// TwinCAT 3 PLC project CNM_RecipeHandling
// Title: CNM_RecipeHandling
// Company: ekvip automation GmbH
// Author: tsch
// ProjectVersion: 0.1.1.0
// Description: This is a TwinCAT 3 library for recipe handling and machine settings. It is intended to be used with CNM HMI framework to store and load parameters.
// ProgramVersion: 3.1.4026.19
// libraries:
//   Tc2_Utilities, * (Beckhoff Automation GmbH)
// project tree:
//   Functions/ CalculateVelocity.TcPOU, ConvertAngle.TcPOU, ConvertAngularVelocity.TcPOU, ConvertArea.TcPOU, ConvertDuration.TcPOU, ConvertLength.TcPOU, ConvertVelocity.TcPOU, ConvertPressure.TcPOU, ConvertTemperature.TcPOU, ConvertVolume.TcPOU, ConvertWeight.TcPOU, FastPow10.TcPOU
//   Functions/Helper/ CheckValueIsANumber.TcPOU
//   Project Information/ F_GetCompany.TcPOU, F_GetTitle.TcPOU, F_GetVersion.TcPOU
//   Types/ Angle.TcDUT, AngularVelocity.TcDUT, Area.TcDUT, BaseParameter.TcDUT, Duration.TcDUT, Length.TcDUT, MetricParameter.TcDUT, Pressure.TcDUT, SiDefaultParameter.TcDUT, Temperature.TcDUT, Velocity.TcDUT, Volume.TcDUT, Weight.TcDUT
//   Types/Units/ AngleUnit.TcDUT, AreaUnit.TcDUT, LengthUnit.TcDUT, DurationUnit.TcDUT, MetricPrefixes.TcDUT, PressureUnit.TcDUT, TemperatureUnit.TcDUT, UnitString.TcDUT, VolumeUnit.TcDUT, WeightUnit.TcDUT
//   Version/ Global_Version.TcGVL

// ---- Types/Angle.TcDUT
(*

## Short summary

A datatype for angles based on angular units. It can be converted to other units with the function CNM_RecipeHandling.ConvertAngle.

.. <legal notes>

legal notes
=================
| SPDX-FileCopyrightText: © 2025 ekvip automation GmbH <info@ekvip.de>
| SPDX-License-Identifier: Apache-2.0
| For details check: Apache-2.0_

.. _Apache-2.0: https://www.apache.org/licenses/LICENSE-2.0

.. </legal notes>	

*)

TYPE Angle EXTENDS BaseParameter:
STRUCT
	(* the angular unit *)
	unit :AngleUnit := AngleUnit.RADIANS;
END_STRUCT
END_TYPE

// ---- Types/AngularVelocity.TcDUT
(*

## Short summary

A datatype for angular velocities based on physical units.

.. <legal notes>

legal notes
=================
| SPDX-FileCopyrightText: © 2025 ekvip automation GmbH <info@ekvip.de>
| SPDX-License-Identifier: Apache-2.0
| For details check: Apache-2.0_

.. _Apache-2.0: https://www.apache.org/licenses/LICENSE-2.0

.. </legal notes>	

*)

TYPE AngularVelocity EXTENDS BaseParameter:
STRUCT
	angularDistanceUnit :AngleUnit := AngleUnit.TURNS;
	timeUnit :DurationUnit := DurationUnit.MINUTE;
	timePrefix :MetricPrefixes := MetricPrefixes.NONE;
END_STRUCT
END_TYPE

// ---- Types/Area.TcDUT
(*

## Short summary

A datatype for areas based on physical units. It can be converted to other units with the function CNM_RecipeHandling.ConvertArea. 

.. <legal notes>

legal notes
=================
| SPDX-FileCopyrightText: © 2025 ekvip automation GmbH <info@ekvip.de>
| SPDX-License-Identifier: Apache-2.0
| For details check: Apache-2.0_

.. _Apache-2.0: https://www.apache.org/licenses/LICENSE-2.0

.. </legal notes>	

*)

TYPE Area EXTENDS MetricParameter:
STRUCT
	(* the area unit *)
	unit :AreaUnit := AreaUnit.SQUARE_METER;
END_STRUCT
END_TYPE

// ---- Types/BaseParameter.TcDUT
(*

## Short summary

A basic datatype for physical parameters. It has just a value. 

.. <legal notes>

legal notes
=================
| SPDX-FileCopyrightText: © 2025 ekvip automation GmbH <info@ekvip.de>
| SPDX-License-Identifier: Apache-2.0
| For details check: Apache-2.0_

.. _Apache-2.0: https://www.apache.org/licenses/LICENSE-2.0

.. </legal notes>	

*)

TYPE BaseParameter :
STRUCT
	value :LREAL := 0.0;
END_STRUCT
END_TYPE

// ---- Types/Duration.TcDUT
(*

## Short summary

A datatype for durations based on physical time units. It can be converted to other units with the function CNM_RecipeHandling.ConvertDuration. 

.. <legal notes>

legal notes
=================
| SPDX-FileCopyrightText: © 2025 ekvip automation GmbH <info@ekvip.de>
| SPDX-License-Identifier: Apache-2.0
| For details check: Apache-2.0_

.. _Apache-2.0: https://www.apache.org/licenses/LICENSE-2.0

.. </legal notes>	

*)

TYPE Duration EXTENDS MetricParameter :
STRUCT
	(* the time unit *)
	unit :DurationUnit := DurationUnit.SECONDS;
END_STRUCT
END_TYPE

// ---- Types/Length.TcDUT
(*

## Short summary

A datatype for distances based on physical length units. It can be converted to other units with the function CNM_RecipeHandling.ConvertLength. 

.. <legal notes>

legal notes
=================
| SPDX-FileCopyrightText: © 2025 ekvip automation GmbH <info@ekvip.de>
| SPDX-License-Identifier: Apache-2.0
| For details check: Apache-2.0_

.. _Apache-2.0: https://www.apache.org/licenses/LICENSE-2.0

.. </legal notes>	

*)

TYPE Length EXTENDS MetricParameter:
STRUCT
	(* the length unit *)
	unit :LengthUnit := LengthUnit.METER;
END_STRUCT
END_TYPE

// ---- Types/MetricParameter.TcDUT
(*

## Short summary

A basic datatype for metrical physical parameters. It extends the CNM_RecipeHandling.BaseParameter with a metric prefix. 

.. <legal notes>

legal notes
=================
| SPDX-FileCopyrightText: © 2025 ekvip automation GmbH <info@ekvip.de>
| SPDX-License-Identifier: Apache-2.0
| For details check: Apache-2.0_

.. _Apache-2.0: https://www.apache.org/licenses/LICENSE-2.0

.. </legal notes>	

*)

TYPE MetricParameter EXTENDS BaseParameter :
STRUCT
	prefix :MetricPrefixes := MetricPrefixes.NONE;
END_STRUCT
END_TYPE

// ---- Types/Pressure.TcDUT
(*

## Short summary

A datatype for pressures based on physical units. It can be converted to other units with the function CNM_RecipeHandling.ConvertPressure. 

.. <legal notes>

legal notes
=================
| SPDX-FileCopyrightText: © 2025 ekvip automation GmbH <info@ekvip.de>
| SPDX-License-Identifier: Apache-2.0
| For details check: Apache-2.0_

.. _Apache-2.0: https://www.apache.org/licenses/LICENSE-2.0

.. </legal notes>	

*)

TYPE Pressure EXTENDS MetricParameter :
STRUCT
	unit :PressureUnit := PressureUnit.PASCAL;
END_STRUCT
END_TYPE

// ---- Types/SiDefaultParameter.TcDUT
(*

## Short summary

A datatype for temperatures based on temperature scales. It can be converted to other units with the function CNM_RecipeHandling.ConvertTemperature. 

.. <legal notes>

legal notes
=================
| SPDX-FileCopyrightText: © 2025 ekvip automation GmbH <info@ekvip.de>
| SPDX-License-Identifier: Apache-2.0
| For details check: Apache-2.0_

.. _Apache-2.0: https://www.apache.org/licenses/LICENSE-2.0

.. </legal notes>	

*)

TYPE SiDefaultParameter EXTENDS MetricParameter :
STRUCT
	unit :UnitString;
END_STRUCT
END_TYPE

// ---- Types/Temperature.TcDUT
(*

## Short summary

A datatype for temperatures based on temperature scales. It can be converted to other units with the function CNM_RecipeHandling.ConvertTemperature. 

.. <legal notes>

legal notes
=================
| SPDX-FileCopyrightText: © 2025 ekvip automation GmbH <info@ekvip.de>
| SPDX-License-Identifier: Apache-2.0
| For details check: Apache-2.0_

.. _Apache-2.0: https://www.apache.org/licenses/LICENSE-2.0

.. </legal notes>	

*)

TYPE Temperature EXTENDS BaseParameter:
STRUCT
	(* the temperature scale *)
	unit :TemperatureUnit := TemperatureUnit.KELVIN;
END_STRUCT
END_TYPE

// ---- Types/Units/AngleUnit.TcDUT
(*

## Short summary

This enumeration contains common angular units including radians, degrees, arc minutes, and arc seconds.

.. <legal notes>

legal notes
=================
| SPDX-FileCopyrightText: © 2025 ekvip automation GmbH <info@ekvip.de>
| SPDX-License-Identifier: Apache-2.0
| For details check: Apache-2.0_

.. _Apache-2.0: https://www.apache.org/licenses/LICENSE-2.0

.. </legal notes>	

*)

{attribute 'qualified_only'}
{attribute 'to_string'}
TYPE AngleUnit :
(
	RADIANS := 0,
	DEGREES,
	ARC_MINUTES,
	ARC_SECONDS,
	GRADIANS,
	TURNS
);
END_TYPE

// ---- Types/Units/AreaUnit.TcDUT
(*

## Short summary

This enumeration contains common physical area units.

.. <legal notes>

legal notes
=================
| SPDX-FileCopyrightText: © 2025 ekvip automation GmbH <info@ekvip.de>
| SPDX-License-Identifier: Apache-2.0
| For details check: Apache-2.0_

.. _Apache-2.0: https://www.apache.org/licenses/LICENSE-2.0

.. </legal notes>	

*)
{attribute 'qualified_only'}
{attribute 'to_string'}
TYPE AreaUnit :
(
	SQUARE_METER := 0,
	US_SQUARE_INCH,
	US_SQUARE_FOOT,
	US_SQUARE_YARD,
	US_ACRE,
	HECTARE
);
END_TYPE

// ---- Types/Units/LengthUnit.TcDUT
(*

## Short summary

This enumeration contains common physical length units.

.. <legal notes>

legal notes
=================
| SPDX-FileCopyrightText: © 2025 ekvip automation GmbH <info@ekvip.de>
| SPDX-License-Identifier: Apache-2.0
| For details check: Apache-2.0_

.. _Apache-2.0: https://www.apache.org/licenses/LICENSE-2.0

.. </legal notes>	

*)

{attribute 'qualified_only'}
{attribute 'to_string'}
TYPE LengthUnit :
(
	METER := 0,
	US_MIL,
	US_INCH,
	US_FOOT,
	US_YARD,
	US_MILE	
);
END_TYPE

// ---- Types/Units/DurationUnit.TcDUT
(*

## Short summary

This enumeration contains common physical time units.

.. <legal notes>

legal notes
=================
| SPDX-FileCopyrightText: © 2025 ekvip automation GmbH <info@ekvip.de>
| SPDX-License-Identifier: Apache-2.0
| For details check: Apache-2.0_

.. _Apache-2.0: https://www.apache.org/licenses/LICENSE-2.0

.. </legal notes>	

*)

{attribute 'qualified_only'}
{attribute 'to_string'}
TYPE DurationUnit :
(
	SECONDS := 0,
	MINUTE,
	HOUR,
	DAY,
	WEEK	
);
END_TYPE

// ---- Types/Units/MetricPrefixes.TcDUT
(*

## Short summary

This is an enumeration for metric prefixes. The value after an enum entry corresponds to the power of ten of the respective prefix. 

.. <legal notes>

legal notes
=================
| SPDX-FileCopyrightText: © 2025 ekvip automation GmbH <info@ekvip.de>
| SPDX-License-Identifier: Apache-2.0
| For details check: Apache-2.0_

.. _Apache-2.0: https://www.apache.org/licenses/LICENSE-2.0

.. </legal notes>	

*)

{attribute 'qualified_only'}
{attribute 'to_string'}
TYPE MetricPrefixes :
(
	QUECTO := -30,
	RONTO := -27 ,
	YOCTO := -24 ,
	ZEPTO := -21 ,
	ATTO := -18  ,
	FEMTO := -15 ,
	PICO := -12  ,
	NANO := -9   ,
	MICRO := -6  ,
	MILLI := -3  ,
	CENTI := -2  ,
	DECI := -1   ,
	NONE := 0    ,
	DEKA := 1    ,
	HECTO := 2   ,
	KILO := 3    ,
	MEGA := 6    ,
	GIGA := 9    ,
	TERA := 12   ,
	PETA := 15   ,
	EXA := 18    ,
	ZETTA := 21  ,
	YOTTA := 24  ,
	RONNA := 27  ,
	QUETTA := 30 
) INT ;
END_TYPE

// ---- Types/Units/PressureUnit.TcDUT
(*

## Short summary

This enumeration contains common physical pressure units.

.. <legal notes>

legal notes
=================
| SPDX-FileCopyrightText: © 2025 ekvip automation GmbH <info@ekvip.de>
| SPDX-License-Identifier: Apache-2.0
| For details check: Apache-2.0_

.. _Apache-2.0: https://www.apache.org/licenses/LICENSE-2.0

.. </legal notes>	

*)

{attribute 'qualified_only'}
{attribute 'to_string'}
TYPE PressureUnit :
(
	PASCAL := 0,
	BAR,
	(* pound per square inch *)
	PSI
);
END_TYPE

// ---- Types/Units/TemperatureUnit.TcDUT
(*

## Short summary

This enumeration contains common temperature scales.

.. <legal notes>

legal notes
=================
| SPDX-FileCopyrightText: © 2025 ekvip automation GmbH <info@ekvip.de>
| SPDX-License-Identifier: Apache-2.0
| For details check: Apache-2.0_

.. _Apache-2.0: https://www.apache.org/licenses/LICENSE-2.0

.. </legal notes>	

*)

{attribute 'qualified_only'}
{attribute 'to_string'}
TYPE TemperatureUnit :
(
	KELVIN := 0,
	DEGREE_CELSIUS,
	DEGREE_FAHRENHEIT
);
END_TYPE

// ---- Types/Units/UnitString.TcDUT
(*

## Short summary

The UnitString is an alias for a string with a limited amount of characters. 

.. <legal notes>

legal notes
=================
| SPDX-FileCopyrightText: © 2025 ekvip automation GmbH <info@ekvip.de>
| SPDX-License-Identifier: Apache-2.0
| For details check: Apache-2.0_

.. _Apache-2.0: https://www.apache.org/licenses/LICENSE-2.0

.. </legal notes>	

*)

TYPE UnitString : STRING(10); END_TYPE

// ---- Types/Units/VolumeUnit.TcDUT
(*

## Short summary

This enumeration contains common physical volume units.

.. <legal notes>

legal notes
=================
| SPDX-FileCopyrightText: © 2025 ekvip automation GmbH <info@ekvip.de>
| SPDX-License-Identifier: Apache-2.0
| For details check: Apache-2.0_

.. _Apache-2.0: https://www.apache.org/licenses/LICENSE-2.0

.. </legal notes>	

*)

{attribute 'qualified_only'}
{attribute 'strict'}
{attribute 'to_string'}
TYPE VolumeUnit :
(
	CUBIC_METER := 0,
	LITER,
	US_CUBIC_INCH,
	US_CUBIC_FOOT,
	US_CUBIC_YARD,
	US_FLUID_OUNCE,
	US_PINT,
	US_GALLON,
	US_BARREL,
	US_OIL_BARREL,
	US_DRY_PINT,
	US_DRY_GALLON,
	US_DRY_BARREL
);
END_TYPE

// ---- Types/Units/WeightUnit.TcDUT
(*

## Short summary

This enumeration contains common physical weight units. The US units are based on the Avoirdupois measurement system.

.. <legal notes>

legal notes
=================
| SPDX-FileCopyrightText: © 2025 ekvip automation GmbH <info@ekvip.de>
| SPDX-License-Identifier: Apache-2.0
| For details check: Apache-2.0_

.. _Apache-2.0: https://www.apache.org/licenses/LICENSE-2.0

.. </legal notes>	

*)


{attribute 'qualified_only'}
{attribute 'to_string'}
TYPE WeightUnit :
(
	GRAM := 0,
	TON,
	US_GRAIN,
	US_DRAM,
	US_OUNCE,
	US_POUND,
	US_TON
);
END_TYPE

// ---- Types/Velocity.TcDUT
(*

## Short summary

A datatype for velocities based on physical units. It can be converted to other units with the function CNM_RecipeHandling.ConvertVelocity.

.. <legal notes>

legal notes
=================
| SPDX-FileCopyrightText: © 2025 ekvip automation GmbH <info@ekvip.de>
| SPDX-License-Identifier: Apache-2.0
| For details check: Apache-2.0_

.. _Apache-2.0: https://www.apache.org/licenses/LICENSE-2.0

.. </legal notes>	

*)

TYPE Velocity EXTENDS BaseParameter:
STRUCT
	distanceUnit :LengthUnit := LengthUnit.METER;
	distancePrefix :MetricPrefixes := MetricPrefixes.NONE;
	timeUnit :DurationUnit := DurationUnit.SECONDS;
	timePrefix :MetricPrefixes := MetricPrefixes.NONE;
END_STRUCT
END_TYPE

// ---- Types/Volume.TcDUT
(*

## Short summary

A datatype for volumes based on physical units. It can be converted to other units with the function CNM_RecipeHandling.ConvertVolume. 

.. <legal notes>

legal notes
=================
| SPDX-FileCopyrightText: © 2025 ekvip automation GmbH <info@ekvip.de>
| SPDX-License-Identifier: Apache-2.0
| For details check: Apache-2.0_

.. _Apache-2.0: https://www.apache.org/licenses/LICENSE-2.0

.. </legal notes>	

*)

TYPE Volume EXTENDS MetricParameter:
STRUCT
	(* the volume unit *)
	unit :VolumeUnit := VolumeUnit.CUBIC_METER;
END_STRUCT
END_TYPE

// ---- Types/Weight.TcDUT
(*

## Short summary

A datatype for weights based on physical weight units. It can be converted to other units with the function CNM_RecipeHandling.ConvertWeight. 

.. <legal notes>

legal notes
=================
| SPDX-FileCopyrightText: © 2025 ekvip automation GmbH <info@ekvip.de>
| SPDX-License-Identifier: Apache-2.0
| For details check: Apache-2.0_

.. _Apache-2.0: https://www.apache.org/licenses/LICENSE-2.0

.. </legal notes>	

*)

TYPE Weight EXTENDS MetricParameter:
STRUCT
	(* the weight unit *)
	unit :WeightUnit := WeightUnit.GRAM;
END_STRUCT
END_TYPE

// ---- Version/Global_Version.TcGVL
{attribute 'TcGenerated'}
{attribute 'no-analysis'}
{attribute 'linkalways'}
// This function has been automatically generated from the project information.
VAR_GLOBAL CONSTANT
	{attribute 'const_non_replaced'}
	stLibVersion_CNM_RecipeHandling : ST_LibVersion := (iMajor := 0, iMinor := 1, iBuild := 1, iRevision := 0, nFlags := 0, sVersion := '0.1.1.0');
END_VAR

// ---- Functions/CalculateVelocity.TcPOU
(*

## Short summary

This function can be used to calculate a veloctiy from given distance and time deltas.

.. <legal notes>

legal notes
=================
| SPDX-FileCopyrightText: © 2025 ekvip automation GmbH <info@ekvip.de>
| SPDX-License-Identifier: Apache-2.0
| For details check: Apache-2.0_

.. _Apache-2.0: https://www.apache.org/licenses/LICENSE-2.0

.. </legal notes>



**Return:** the calculated velocity in METER per SECOND
	

*)
FUNCTION CalculateVelocity : Velocity
VAR_IN_OUT
	(* the distance to travel *)
	distanceDelta :Length;
	(* the time it needs to travel *)
	timeDelta :Duration; 
END_VAR
VAR
	tmpDistance :Length;
	tmpTime :Duration;
END_VAR

// return if we are not able to calculate
RETURN(
		(timeDelta.value = 0.0) // we cannot divide by zero without destroying the universe
	OR_ELSE 
		NOT CheckValueIsANumber(distanceDelta.value)
	OR_ELSE 
		NOT CheckValueIsANumber(timeDelta.value)
);

IF (	(distanceDelta.unit = LengthUnit.METER)
	AND_THEN
		(distanceDelta.prefix = MetricPrefixes.NONE)
	AND_THEN
		(timeDelta.unit = DurationUnit.SECONDS)
	AND_THEN
		(timeDelta.prefix = MetricPrefixes.NONE)
	)
THEN
	CalculateVelocity.value := distanceDelta.value / timeDelta.value;
ELSE
	tmpDistance := ConvertLength(distanceDelta);
	tmpTime := ConvertDuration(timeDelta);
	CalculateVelocity.value := tmpDistance.value / tmpTime.value;
END_IF

END_FUNCTION

// ---- Functions/Helper/CheckValueIsANumber.TcPOU
(*

## Short summary

This function checks if the given LREAL is a valid number to calculate with.

.. <legal notes>

legal notes
=================
| SPDX-FileCopyrightText: © 2025 ekvip automation GmbH <info@ekvip.de>
| SPDX-License-Identifier: Apache-2.0
| For details check: Apache-2.0_

.. _Apache-2.0: https://www.apache.org/licenses/LICENSE-2.0

.. </legal notes>



**Return:** TRUE if the value is processable, FALSE if NaN or +/-Inf
	
*)

FUNCTION INTERNAL CheckValueIsANumber : BOOL
VAR_INPUT 
	(* the folating point that should be checked *)
	value :LREAL;
END_VAR

CheckValueIsANumber := (NOT Tc2_Utilities.LrealIsNaN(value)) AND_THEN Tc2_Utilities.LrealIsFinite(value);

END_FUNCTION

// ---- Functions/ConvertLength.TcPOU
(*

## Short summary

This function can be used to convert distances from one physical length unit into another. The value will change corresponding to the conversion.
**Example:**  
1 m =  39.3701 inches = 3.28084167 feet = 1.093613889 yard = 0.00062137 miles

.. <legal notes>

legal notes
=================
| SPDX-FileCopyrightText: © 2025 ekvip automation GmbH <info@ekvip.de>
| SPDX-License-Identifier: Apache-2.0
| For details check: Apache-2.0_

.. _Apache-2.0: https://www.apache.org/licenses/LICENSE-2.0

.. </legal notes>



**Return:** CNM_RecipeHandling.Length: a copy of the given length converted into the desired unit
	

*)

FUNCTION ConvertLength : Length
VAR_IN_OUT CONSTANT
	(* the length that should be converted *)
	lengthToConvert :Length;
END_VAR
VAR_INPUT
	(* the physical length unit it should be converted to *)
	convertTo :LengthUnit := LengthUnit.METER;
	(* the metrical prefix (for SI units) *)
	resultPrefix :MetricPrefixes := MetricPrefixes.NONE;
END_VAR
VAR
	factor :LREAL;
	exponent :INT := 1;
END_VAR
VAR CONSTANT
	(* length convertions related to meter *)
	LENGTHS : ARRAY[LengthUnit.METER..LengthUnit.US_MILE] OF LREAL := [1.0, 2.54E-5, 0.0254, 0.3048, 0.9144, 1609.34];
END_VAR

factor := LENGTHS[lengthToConvert.unit] / LENGTHS[convertTo];
exponent := lengthToConvert.prefix - resultPrefix;
ConvertLength.prefix := resultPrefix;
ConvertLength.unit := convertTo;
IF CheckValueIsANumber(lengthToConvert.value) THEN
	ConvertLength.value := lengthToConvert.value * factor * FastPow10(exponent);
ELSE
	ConvertLength.value := lengthToConvert.value;
END_IF

END_FUNCTION

// ---- Functions/FastPow10.TcPOU
(*

## Short summary

This function calculates the power of ten with the given exponent efficiently using exponentiation by squaring for exponents > 3. 
It supports both positive and negative integer exponents.

.. <legal notes>

legal notes
=================
| SPDX-FileCopyrightText: © 2025 ekvip automation GmbH <info@ekvip.de>
| SPDX-License-Identifier: Apache-2.0
| For details check: Apache-2.0_

.. _Apache-2.0: https://www.apache.org/licenses/LICENSE-2.0

.. </legal notes>



**Return:** the power of 10 for the given exponent as LREAL 
*)

FUNCTION FastPow10 : LREAL
VAR_INPUT
	(* The exponent to which the base is raised. Can be positive or negative. *)
	exponent :INT;
END_VAR
VAR
	calcExponent :WORD := 1;
	mask :INT;
	base :LREAL := 10.0;
END_VAR
VAR CONSTANT
	SMALL_POWERS : ARRAY[0..3] OF LREAL := [1.0, 10.0, 100.0, 1000.0];
END_VAR

// get absolute value of exponent
mask := SHR(exponent, SIZEOF(INT)*8 - 1);
{warning disable C0195} // conversion from INT to UINT desired, this is an ABS(exponent)
calcExponent := (exponent + mask) XOR mask;
{warning restore C0195}
// for small exponents use the mapping
IF (calcExponent <= 3) THEN
	FastPow10 := SMALL_POWERS[calcExponent];
ELSE
// with great power comes great potential for optimization lol :) 
	// exponentation by squaring, needs less multiplications then EXPT for exponents > 3
	FastPow10 := 1.0;
	WHILE (calcExponent > 0) DO
		IF ((calcExponent AND 1) = 1) THEN
			FastPow10 := FastPow10 * base;	
		END_IF
		base := base * base;
		calcExponent := SHR(calcExponent,1); 
	END_WHILE
END_IF
// inverse it if exponent was negative
FastPow10 := SEL((exponent > 0), 1 / FastPow10, FastPow10);

END_FUNCTION

// ---- Functions/ConvertDuration.TcPOU
(*

## Short summary

This function can be used to convert durations from one physical time unit into another. The value will change corresponding to the conversion.
**Example:**  
15 s =  0.25 min = 0.00416667 h = 0.00017361125 days = 2.4801607143e-5 weeks 

.. <legal notes>

legal notes
=================
| SPDX-FileCopyrightText: © 2025 ekvip automation GmbH <info@ekvip.de>
| SPDX-License-Identifier: Apache-2.0
| For details check: Apache-2.0_

.. _Apache-2.0: https://www.apache.org/licenses/LICENSE-2.0

.. </legal notes>



**Return:** CNM_RecipeHandling.Duration: a copy of the given duration converted into the desired unit
	

*)

FUNCTION ConvertDuration : Duration
VAR_IN_OUT CONSTANT
	(* the duration that should be converted *)
	durationToConvert :Duration;
END_VAR
VAR_INPUT
	(* the physical time unit it should be converted to *)
	convertTo :DurationUnit := DurationUnit.SECONDS;
	(* the metrical prefix (for SI units) *)
	resultPrefix :MetricPrefixes := MetricPrefixes.NONE;
END_VAR
VAR
	factor :LREAL;
	exponent :INT := 1;
END_VAR
VAR CONSTANT
	(* duration convertions related to seconds *)
	DURATIONS : ARRAY[DurationUnit.SECONDS..DurationUnit.WEEK] OF LREAL := [1.0, 60.0, 3600.0, 86400.0, 604800.0];
END_VAR

factor := DURATIONS[durationToConvert.unit] / DURATIONS[convertTo];
exponent := durationToConvert.prefix - resultPrefix;
ConvertDuration.prefix := resultPrefix;
ConvertDuration.unit := convertTo;
IF CheckValueIsANumber(durationToConvert.value) THEN
	ConvertDuration.value := durationToConvert.value * factor * FastPow10(exponent);
ELSE
	ConvertDuration.value := durationToConvert.value;
END_IF

END_FUNCTION

// ---- Functions/ConvertAngle.TcPOU
(*

## Short summary

This function can be used to convert angles from one angular unit into another. The value will change corresponding to the conversion.
**Example:** 
π radians = 180° = 10800' = 648000" = 200 gradians = 0.5 turns

.. <legal notes>

legal notes
=================
| SPDX-FileCopyrightText: © 2025 ekvip automation GmbH <info@ekvip.de>
| SPDX-License-Identifier: Apache-2.0
| For details check: Apache-2.0_

.. _Apache-2.0: https://www.apache.org/licenses/LICENSE-2.0

.. </legal notes>



**Return:** CNM_RecipeHandling.Angle: a copy of the given angle converted into the desired unit
	

*)

FUNCTION ConvertAngle : Angle
VAR_IN_OUT CONSTANT
	(* the angle that should be converted *)
	angleToConvert :Angle;
END_VAR
VAR_INPUT
	(* the angular unit it should be converted to *)
	convertTo :AngleUnit := AngleUnit.RADIANS;
END_VAR
VAR
	factor :LREAL;
END_VAR
VAR CONSTANT
	PI :LREAL := 3.14159265358979323846264338327950288;
	(* angle conversions related to radians (base unit) *)
	ANGLES : ARRAY[AngleUnit.RADIANS..AngleUnit.TURNS] OF LREAL := [
		1.0,								// RADIANS (base unit)
		PI / 180.0,							// DEGREES to radians
		PI / 10800.0,						// ARC_MINUTES to radians
		PI / 648000.0,						// ARC_SECONDS to radians
		PI / 200.0,							// GRADIANS to radians
		2.0 * PI							// TURNS to radians
	];
END_VAR

factor := ANGLES[angleToConvert.unit] / ANGLES[convertTo];
ConvertAngle.unit := convertTo;
IF CheckValueIsANumber(angleToConvert.value) THEN
	ConvertAngle.value := angleToConvert.value * factor;
ELSE
	ConvertAngle.value := angleToConvert.value;
END_IF

END_FUNCTION

// ---- Functions/ConvertAngularVelocity.TcPOU
(*
## Short summary

This function converts angular velocities from one unit into another.
The value is adjusted according to the unit conversion factors.

**Example:**
1 turn/min = 6.28319 rad/min = 0.10472 rad/s = 360 deg/min = 6 deg/s

.. <legal notes>

legal notes
=================
| SPDX-FileCopyrightText: © 2025 ekvip automation GmbH <info@ekvip.de>
| SPDX-License-Identifier: Apache-2.0
| For details check: Apache-2.0_

.. _Apache-2.0: https://www.apache.org/licenses/LICENSE-2.0

.. </legal notes>



**Return:** CNM_RecipeHandling.AngularVelocity: a copy of the given angular velocity converted into the desired unit

*)
FUNCTION ConvertAngularVelocity :AngularVelocity
VAR_IN_OUT CONSTANT
    (* the angular velocity that should be converted *)
    angularVelocityToConvert :AngularVelocity;
END_VAR
VAR_INPUT
    (* the physical angle unit it should be converted to *)
    convertAngleTo :AngleUnit := AngleUnit.TURNS;
    (* the physical time unit it should be converted to *)
    convertTimeTo :DurationUnit := DurationUnit.MINUTE;
    (* the metrical prefix for the time *)
    resultPrefixTime :MetricPrefixes := MetricPrefixes.NONE;
END_VAR
VAR
    factorAngle, factorTime : LREAL;
    exponent : INT := 1;
END_VAR
VAR CONSTANT
	PI :LREAL := 3.14159265358979323846264338327950288;
	(* angle conversions related to radians (base unit) *)
	ANGLES : ARRAY[AngleUnit.RADIANS..AngleUnit.TURNS] OF LREAL := [
		1.0,								// RADIANS (base unit)
		PI / 180.0,							// DEGREES to radians
		PI / 10800.0,						// ARC_MINUTES to radians
		PI / 648000.0,						// ARC_SECONDS to radians
		PI / 200.0,							// GRADIANS to radians
		2.0 * PI							// TURNS to radians
	];
    (* duration conversions related to second *)
    DURATIONS : ARRAY[DurationUnit.SECONDS..DurationUnit.WEEK] OF LREAL := [1.0, 60.0, 3600.0, 86400.0, 604800.0];
END_VAR

(* calculate conversion factors *)
factorAngle := ANGLES[angularVelocityToConvert.angularDistanceUnit] / ANGLES[convertAngleTo];
factorTime := DURATIONS[angularVelocityToConvert.timeUnit] / DURATIONS[convertTimeTo];

(* apply metric prefix scaling, same logic as ConvertVelocity *)
exponent := resultPrefixTime - angularVelocityToConvert.timePrefix;

(* assign target units *)
ConvertAngularVelocity.angularDistanceUnit := convertAngleTo;
ConvertAngularVelocity.timeUnit := convertTimeTo;
ConvertAngularVelocity.timePrefix := resultPrefixTime;

(* perform conversion if the value is valid *)
IF CheckValueIsANumber(angularVelocityToConvert.value) THEN
	ConvertAngularVelocity.value := angularVelocityToConvert.value * factorAngle / factorTime * FastPow10(exponent);
ELSE
	ConvertAngularVelocity.value := angularVelocityToConvert.value;
END_IF

END_FUNCTION

// ---- Functions/ConvertArea.TcPOU
(*

## Short summary

This function can be used to convert areas from one physical unit into another. The value will change corresponding to the conversion.
**Example:** 
1 square meter =  1E-6 square kilometer = 1550 square inch = 10.7639 square foot = 1.19599 square yard.

.. <legal notes>

legal notes
=================
| SPDX-FileCopyrightText: © 2025 ekvip automation GmbH <info@ekvip.de>
| SPDX-License-Identifier: Apache-2.0
| For details check: Apache-2.0_

.. _Apache-2.0: https://www.apache.org/licenses/LICENSE-2.0

.. </legal notes>



**Return:** CNM_RecipeHandling.Area: a copy of the given area converted into the desired unit
	
*)

FUNCTION ConvertArea : Area
VAR_IN_OUT CONSTANT
	(* the area that should be converted *)
	areaToConvert :Area;
END_VAR
VAR_INPUT
	(* the physical unit it should be converted to *)
	convertTo :AreaUnit := AreaUnit.SQUARE_METER;
	(* the metrical prefix (for SI units) *)
	resultPrefix :MetricPrefixes := MetricPrefixes.NONE;
END_VAR
VAR
	factor :LREAL;
	exponent :INT := 1;
END_VAR
VAR CONSTANT
	(* area convertions related to squaremeter: square inch, square foot, square yard, acre *)
	AREAS : ARRAY[AreaUnit.SQUARE_METER..AreaUnit.HECTARE] OF LREAL := [
		1.0,  			// in square meter
		0.00064516, 	// in square inch
		0.0929034, 		// in square foot
		0.83612736, 	// in square yard
		4046.873,		// in us acre,
		10000.0			// in hectare
	];
	(* mapping that returns the correct exponentiation factor for sqared or linear units *)
	UNIT_SPECIFIC_FACTOR :ARRAY[AreaUnit.SQUARE_METER..AreaUnit.HECTARE] OF USINT := [	
		2,  	// in square meter
		2, 		// in square inch
		2, 		// in square foot
		2, 		// in square yard
		1, 		// in us acre,
		1		// in hectare
	]; 
END_VAR

factor := AREAS[areaToConvert.unit] / AREAS[convertTo];
exponent := ((UNIT_SPECIFIC_FACTOR[areaToConvert.unit] * areaToConvert.prefix) 
			- ( UNIT_SPECIFIC_FACTOR[convertTo] * resultPrefix));
ConvertArea.prefix := resultPrefix;
ConvertArea.unit := convertTo;
IF CheckValueIsANumber(areaToConvert.value) THEN
	ConvertArea.value := areaToConvert.value * factor * FastPow10(exponent);
ELSE
	ConvertArea.value := areaToConvert.value;
END_IF

END_FUNCTION

// ---- Functions/ConvertVelocity.TcPOU
(*

## Short summary

This function can be used to convert velocities from one unit into another. The value will change corresponding to the conversion.
**Example:**  
1 m/s =  0.001 km/s = 3.6 km/h = 2.23694 miles/h

.. <legal notes>

legal notes
=================
| SPDX-FileCopyrightText: © 2025 ekvip automation GmbH <info@ekvip.de>
| SPDX-License-Identifier: Apache-2.0
| For details check: Apache-2.0_

.. _Apache-2.0: https://www.apache.org/licenses/LICENSE-2.0

.. </legal notes>



**Return:** CNM_RecipeHandling.Velocity: a copy of the given velocity converted into the desired unit
	

*)

FUNCTION ConvertVelocity : Velocity
VAR_IN_OUT CONSTANT
	(* the velocity that should be converted *)
	velocityToConvert :Velocity;
END_VAR
VAR_INPUT
	(* the physical length unit it should be converted to *)
	convertDistanceTo :LengthUnit := LengthUnit.METER;
	(* the physical time unit it should be converted to *)
	convertTimeTo :DurationUnit := DurationUnit.SECONDS;
	(* the metrical prefix for the distance (for SI units) *)
	resultPrefixDistance :MetricPrefixes := MetricPrefixes.NONE;
	(* the metrical prefix for the time *)
	resultPrefixTime :MetricPrefixes := MetricPrefixes.NONE;
END_VAR
VAR
	factorLength, factorTime :LREAL;
	exponent :INT := 1;
END_VAR
VAR CONSTANT
	(* length convertions related to meter *)
	LENGTHS : ARRAY[LengthUnit.METER..LengthUnit.US_MILE] OF LREAL := [1.0, 2.54E-5, 0.0254, 0.3048, 0.9144, 1609.34];
	(* duration convertions related to seconds *)
	DURATIONS : ARRAY[DurationUnit.SECONDS..DurationUnit.WEEK] OF LREAL := [1.0, 60.0, 3600.0, 86400.0, 604800.0];
END_VAR

factorLength := LENGTHS[velocityToConvert.distanceUnit] / LENGTHS[convertDistanceTo];
factorTime := DURATIONS[velocityToConvert.timeUnit] / DURATIONS[convertTimeTo];
exponent := velocityToConvert.distancePrefix - resultPrefixDistance - velocityToConvert.timePrefix + resultPrefixTime;
ConvertVelocity.distanceUnit := convertDistanceTo;
ConvertVelocity.distancePrefix := resultPrefixDistance;
ConvertVelocity.timeUnit := convertTimeTo;
ConvertVelocity.timePrefix := resultPrefixTime;
IF CheckValueIsANumber(velocityToConvert.value) THEN
	ConvertVelocity.value := velocityToConvert.value * factorLength/factorTime * FastPow10(exponent);
ELSE
	ConvertVelocity.value := velocityToConvert.value;
END_IF

END_FUNCTION

// ---- Functions/ConvertPressure.TcPOU
(*

## Short summary

This function can be used to convert pressures from one physical pressure unit into another. The value will change corresponding to the conversion.
**Example:**  
1 Pa =  0.00001 Bar = 0.000145038 Psi

.. <legal notes>

legal notes
=================
| SPDX-FileCopyrightText: © 2025 ekvip automation GmbH <info@ekvip.de>
| SPDX-License-Identifier: Apache-2.0
| For details check: Apache-2.0_

.. _Apache-2.0: https://www.apache.org/licenses/LICENSE-2.0

.. </legal notes>



**Return:** CNM_RecipeHandling.Pressure: a copy of the given pressure converted into the desired unit
	

*)

FUNCTION ConvertPressure : Pressure
VAR_IN_OUT CONSTANT
	(* the pressure that should be converted *)
	pressureToConvert :Pressure;
END_VAR
VAR_INPUT
	(* the physical pressure unit it should be converted to *)
	convertTo :PressureUnit := PressureUnit.PASCAL;
	(* the metrical prefix (for SI units) *)
	resultPrefix :MetricPrefixes := MetricPrefixes.NONE;
END_VAR
VAR
	factor :LREAL;
	exponent :INT := 1;
END_VAR
VAR CONSTANT
	(* length convertions related to pascal *)
	PRESSURES : ARRAY[PressureUnit.PASCAL..PressureUnit.PSI] OF LREAL := [1.0, 100000.0, 6894.76];
END_VAR

factor := PRESSURES[pressureToConvert.unit] / PRESSURES[convertTo];
exponent := pressureToConvert.prefix - resultPrefix;
ConvertPressure.prefix := resultPrefix;
ConvertPressure.unit := convertTo;
IF CheckValueIsANumber(pressureToConvert.value) THEN
	ConvertPressure.value := pressureToConvert.value * factor * FastPow10(exponent);	
ELSE
	ConvertPressure.value := pressureToConvert.value;
END_IF

END_FUNCTION

// ---- Functions/ConvertTemperature.TcPOU
(*

## Short summary

This function can be used to convert temperatures from one temperature scale into another. The value will change corresponding to the conversion.
**Example:**  
300 K = 26.85°C = 80.33 °F

.. <legal notes>

legal notes
=================
| SPDX-FileCopyrightText: © 2025 ekvip automation GmbH <info@ekvip.de>
| SPDX-License-Identifier: Apache-2.0
| For details check: Apache-2.0_

.. _Apache-2.0: https://www.apache.org/licenses/LICENSE-2.0

.. </legal notes>



**Return:** CNM_RecipeHandling.Temprature: a copy of the given temperature converted into the desired scale
	

*)

FUNCTION ConvertTemperature : Temperature
VAR_IN_OUT CONSTANT
	(* the temperature that should be converted *)
	temperatureToConvert :Temperature;
END_VAR
VAR_INPUT
	(* the temperature scale unit it should be converted to *)
	convertTo :TemperatureUnit := TemperatureUnit.KELVIN;
END_VAR
VAR CONSTANT
	CELSIUS_OFFSET :LREAL := 273.15;
	FAHRENHEIT_OFFSET :LREAL := 32.0;
	FAHRENHEIT_FACTOR :LREAL := 1.8;
END_VAR

ConvertTemperature.unit := convertTo;
IF (NOT CheckValueIsANumber(temperatureToConvert.value)) THEN
	ConvertTemperature.value := temperatureToConvert.value;
	RETURN;
END_IF

CASE temperatureToConvert.unit OF
TemperatureUnit.KELVIN:
	CASE convertTo OF
	TemperatureUnit.DEGREE_CELSIUS:
		ConvertTemperature.value := temperatureToConvert.value - CELSIUS_OFFSET;
	TemperatureUnit.DEGREE_FAHRENHEIT:
		ConvertTemperature.value := ((temperatureToConvert.value - CELSIUS_OFFSET) * FAHRENHEIT_FACTOR) + FAHRENHEIT_OFFSET;
	ELSE
		ConvertTemperature.value := temperatureToConvert.value;
	END_CASE
TemperatureUnit.DEGREE_CELSIUS:
	CASE convertTo OF
	TemperatureUnit.KELVIN:
		ConvertTemperature.value := temperatureToConvert.value + CELSIUS_OFFSET;
	TemperatureUnit.DEGREE_FAHRENHEIT:
		ConvertTemperature.value := (temperatureToConvert.value * FAHRENHEIT_FACTOR) + FAHRENHEIT_OFFSET;
	ELSE
		ConvertTemperature.value := temperatureToConvert.value;
	END_CASE
TemperatureUnit.DEGREE_FAHRENHEIT:
	CASE convertTo OF
	TemperatureUnit.KELVIN:
		ConvertTemperature.value := (temperatureToConvert.value - FAHRENHEIT_OFFSET)/FAHRENHEIT_FACTOR + CELSIUS_OFFSET;
	TemperatureUnit.DEGREE_CELSIUS:
		ConvertTemperature.value := (temperatureToConvert.value - FAHRENHEIT_OFFSET)/FAHRENHEIT_FACTOR;
	ELSE
		ConvertTemperature.value := temperatureToConvert.value;
	END_CASE
ELSE
	ConvertTemperature.value := temperatureToConvert.value;
END_CASE

END_FUNCTION

// ---- Functions/ConvertVolume.TcPOU
(*

## Short summary

This function can be used to convert volumes from one physical unit into another. The value will change corresponding to the conversion.
**Example:**  
15 cubic meter = 15000 liter = 915356 cubic inches = 529.7199 cubic feet = 19.6193 cubic yard = 507211.39315817 fluid ounces = 31700.7121 cubic pints = 1816.17 dry pints

.. <legal notes>

legal notes
=================
| SPDX-FileCopyrightText: © 2025 ekvip automation GmbH <info@ekvip.de>
| SPDX-License-Identifier: Apache-2.0
| For details check: Apache-2.0_

.. _Apache-2.0: https://www.apache.org/licenses/LICENSE-2.0

.. </legal notes>



**Return:** CNM_RecipeHandling.Volume: a copy of the given volume converted into the desired unit

*)

FUNCTION ConvertVolume :Volume
VAR_IN_OUT CONSTANT
	(* the volume that should be converted *)
	volumeToConvert :Volume;
END_VAR
VAR_INPUT
	(* the physical volume unit it should be converted to *)
	convertTo :VolumeUnit := VolumeUnit.CUBIC_METER;
	(* the metrical prefix (for SI units) *)
	resultPrefix :MetricPrefixes := MetricPrefixes.NONE;
END_VAR
VAR
	factor :LREAL;
	exponent :INT := 1;
END_VAR
VAR CONSTANT
	(* area convertions related to cubicmeter: square inch, square foot, square yard, acre *)
	VOLUMES : ARRAY[VolumeUnit.CUBIC_METER..VolumeUnit.US_DRY_BARREL ] OF LREAL := [ 
		1.0,  			// in cubic meter
		0.001, 			// in liter
		1.6387E-5, 		// in cubic inch
		0.0283168, 		// in cubic foot
		0.764555, 		// in cubic yard
		2.9573549E-5, 	// in fluid ounce 
		0.000473176, 	// in us pint
		0.00378541, 	// in us gallon
		0.11924, 		// in us barrel
		0.1589872949,		// in us oil barrel
		0.00055061, 	// in us dry pint
		0.00440488, 	// in us dry gallon
		0.115627 		// in us dry barrel
	];
	(* mapping that returns the correct exponentiation factor for cubic or linear units *)
	UNIT_SPECIFIC_FACTOR :ARRAY[VolumeUnit.CUBIC_METER..VolumeUnit.US_DRY_BARREL] OF USINT := [	
		3,  		// in cubic meter
		1, 		// in liter
		3, 		// in cubic inch
		3, 		// in cubic foot
		3, 		// in cubic yard
		1, 		// in fluid ounce
		1, 		// in us pint
		1, 		// in us gallon
		1, 		// in us barrel
		1, 		// in us oil barrel
		1, 		// in us dry pint
		1, 		// in us dry gallon
		1 		// in us dry barrel
	]; 
END_VAR

factor := VOLUMES[volumeToConvert.unit] / VOLUMES[convertTo];
exponent := ((UNIT_SPECIFIC_FACTOR[volumeToConvert.unit] * volumeToConvert.prefix) 
			- (UNIT_SPECIFIC_FACTOR[convertTo] *  resultPrefix));
ConvertVolume.prefix := resultPrefix;
ConvertVolume.unit := convertTo;
IF CheckValueIsANumber(volumeToConvert.value) THEN
	ConvertVolume.value := volumeToConvert.value * factor * FastPow10(exponent);
ELSE
	ConvertVolume.value := volumeToConvert.value;
END_IF

END_FUNCTION

// ---- Functions/ConvertWeight.TcPOU
(*

## Short summary

This function can be used to convert weights from one physical weight unit into another. The value will change corresponding to the conversion.
**Example:**  
10 g =  154,324 US grain = 0.35274 US ounces = 0.564382 US dram = 0.01 kg = 0.00220462 US pounds

.. <legal notes>

legal notes
=================
| SPDX-FileCopyrightText: © 2025 ekvip automation GmbH <info@ekvip.de>
| SPDX-License-Identifier: Apache-2.0
| For details check: Apache-2.0_

.. _Apache-2.0: https://www.apache.org/licenses/LICENSE-2.0

.. </legal notes>



**Return:** CNM_RecipeHandling.Weight: a copy of the given weight converted into the desired unit
	

*)

FUNCTION ConvertWeight : Weight
VAR_IN_OUT CONSTANT
	(* the weight that should be converted *)
	weightToConvert :Weight;
END_VAR
VAR_INPUT
	(* the physical weight unit it should be converted to *)
	convertTo :WeightUnit := WeightUnit.GRAM;
	(* the metrical prefix (for SI units) *)
	resultPrefix :MetricPrefixes := MetricPrefixes.NONE;
END_VAR
VAR
	factor :LREAL;
	exponent :INT := 1;
END_VAR
VAR CONSTANT
	(* weight convertions related to gram: gram, ton, US grain, US dram, US ounce, US pound, US ton *)
	WEIGTHS : ARRAY[WeightUnit.GRAM..WeightUnit.US_TON] OF LREAL := [1.0, 1.0E6, 64.79891E-3, 1.771845195, 28.349523125, 453.59237, 907.18474E3 ];
END_VAR

factor := WEIGTHS[weightToConvert.unit] / WEIGTHS[convertTo];
exponent := weightToConvert.prefix - resultPrefix;
ConvertWeight.prefix := resultPrefix;
ConvertWeight.unit := convertTo;
IF CheckValueIsANumber(weightToConvert.value) THEN
	ConvertWeight.value := weightToConvert.value * factor * FastPow10(exponent);
ELSE
	ConvertWeight.value := weightToConvert.value;
END_IF

END_FUNCTION

// ---- Project Information/F_GetCompany.TcPOU
// This function has been automatically generated from the project information.
{attribute 'signature_flag' := '1073741824'}
{attribute 'TcGenerated'}
{attribute 'no-analysis'}
FUNCTION F_GetCompany : WSTRING
VAR_INPUT
	
END_VAR

F_GetCompany := "ekvip automation GmbH";

END_FUNCTION

// ---- Project Information/F_GetTitle.TcPOU
// This function has been automatically generated from the project information.
{attribute 'signature_flag' := '1073741824'}
{attribute 'TcGenerated'}
{attribute 'no-analysis'}
FUNCTION F_GetTitle : WSTRING
VAR_INPUT
	
END_VAR

F_GetTitle := "CNM_RecipeHandling";

END_FUNCTION

// ---- Project Information/F_GetVersion.TcPOU
// This function has been automatically generated from the project information.
{attribute 'signature_flag' := '1073741824'}
{attribute 'TcGenerated'}
{attribute 'no-analysis'}
FUNCTION F_GetVersion : ST_LibVersion
VAR_INPUT
	
END_VAR

F_GetVersion.iMajor := 0;
F_GetVersion.iMinor := 1;
F_GetVersion.iBuild := 1;
F_GetVersion.iRevision := 0;
F_GetVersion.sVersion := '0.1.1.0';
F_GetVersion.nFlags := 0;

END_FUNCTION
